FUNCTION_BLOCK Manual
VAR_INPUT
END_VAR

VAR_OUTPUT
END_VAR

VAR
	motorSelect: Multiplexer;
	EdgeDetectionRedButton: EdgeDetection;
	TIMER: TIMER;
	
	CountDown: CTUD;
	EdgeDetectionCD: BOOL;
	dropTimer: TON;
	rotateTimer: TON;
	stretchTimer: TON;
	clawTimer: TON;
	CounterDol: CTUD;
	visina: WORD;
	CounterCCW: CTUD;
	rotacija: WORD;
	CounterRazteg: CTUD;
	dolzina: WORD;
	CounterKlesce: CTUD;
	prijem: WORD;
	CounterVisina: CTUD;
END_VAR

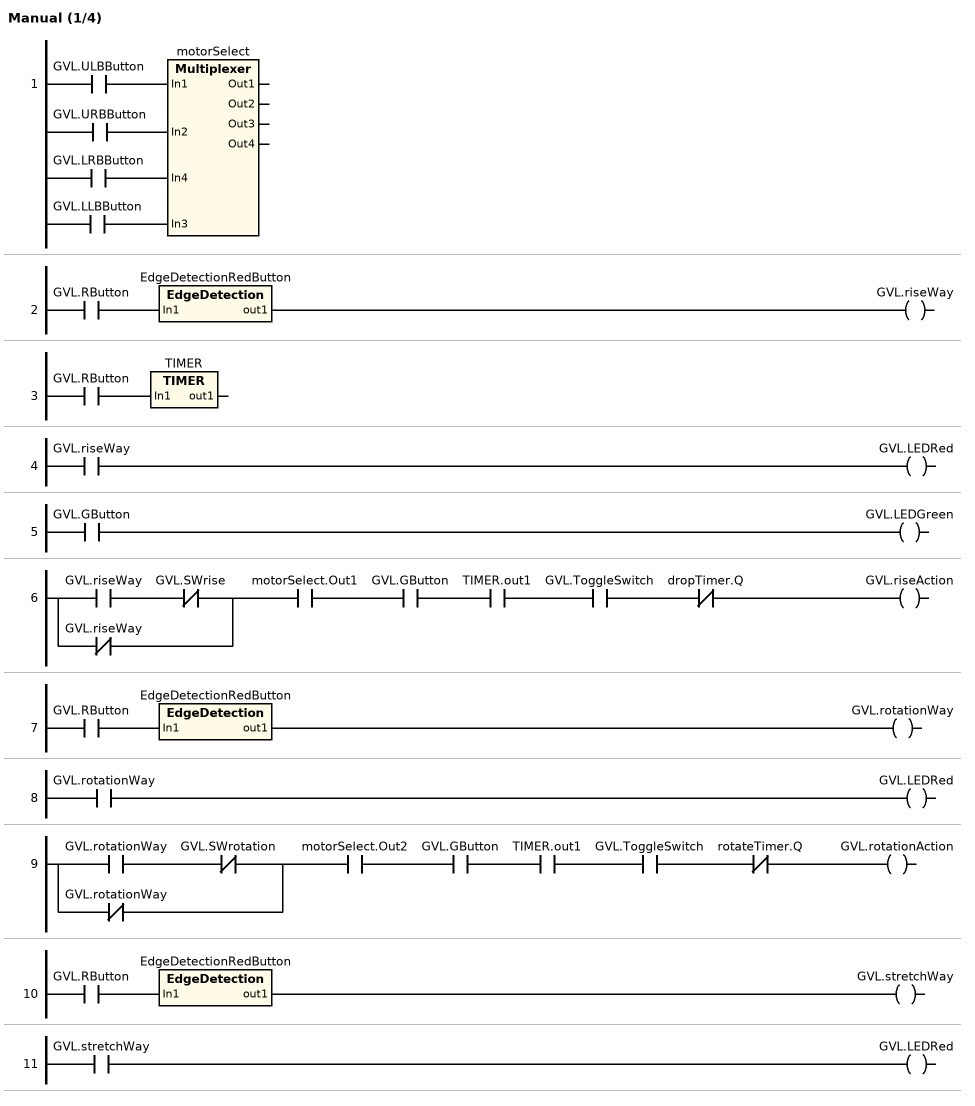
// NETWORK 1
motorSelect(In1 := GVL.ULBButton, In2 := GVL.URBButton, In4 := GVL.LRBButton, In3 := GVL.LLBButton); // Multiplexer

// NETWORK 2
EdgeDetectionRedButton(In1 := GVL.RButton); // EdgeDetection
GVL.riseWay := EdgeDetectionRedButton.out1;

// NETWORK 3
TIMER(In1 := GVL.RButton);

// NETWORK 4
GVL.LEDRed := GVL.riseWay;

// NETWORK 5
GVL.LEDGreen := GVL.GButton;

// NETWORK 6
GVL.riseAction := (GVL.riseWay AND NOT GVL.SWrise OR NOT GVL.riseWay) AND motorSelect.Out1 AND GVL.GButton AND TIMER.out1 AND GVL.ToggleSwitch AND NOT dropTimer.Q;

// NETWORK 7
EdgeDetectionRedButton(In1 := GVL.RButton); // EdgeDetection
GVL.rotationWay := EdgeDetectionRedButton.out1;

// NETWORK 8
GVL.LEDRed := GVL.rotationWay;

// NETWORK 9
GVL.rotationAction := (GVL.rotationWay AND NOT GVL.SWrotation OR NOT GVL.rotationWay) AND motorSelect.Out2 AND GVL.GButton AND TIMER.out1 AND GVL.ToggleSwitch AND NOT rotateTimer.Q;

// NETWORK 10
EdgeDetectionRedButton(In1 := GVL.RButton); // EdgeDetection
GVL.stretchWay := EdgeDetectionRedButton.out1;

// NETWORK 11
GVL.LEDRed := GVL.stretchWay;

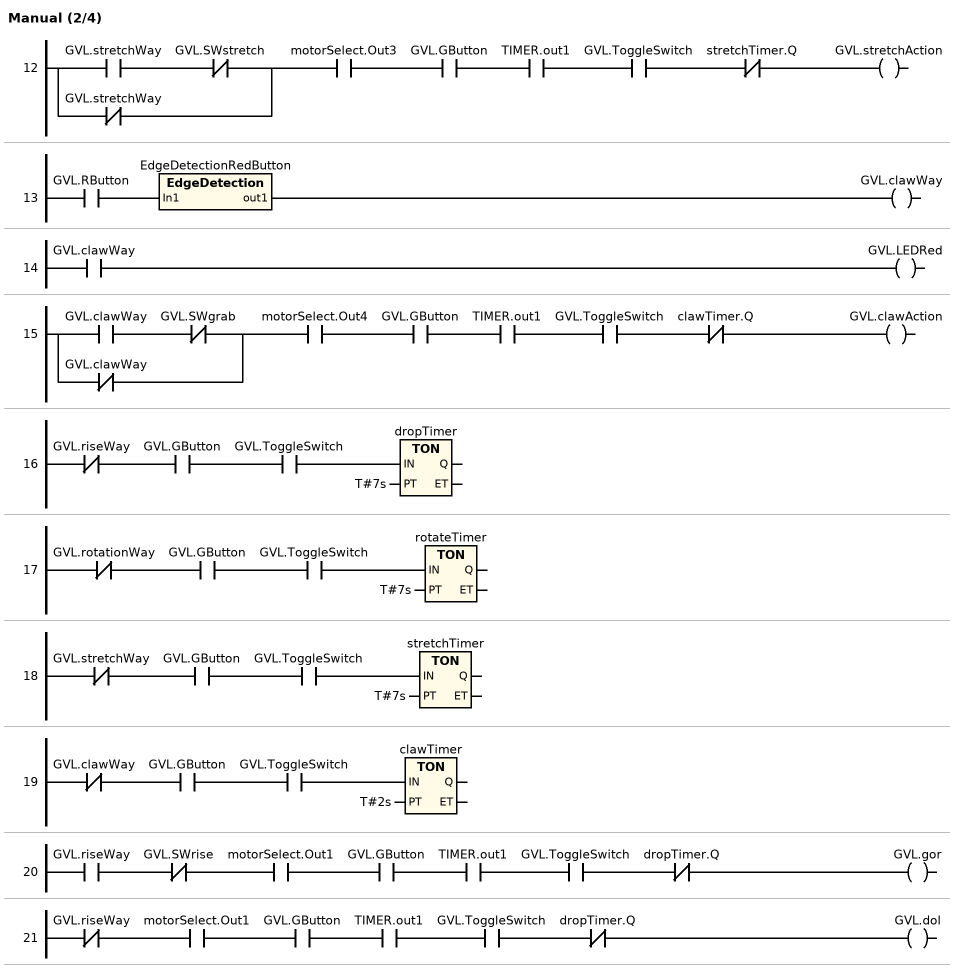
// NETWORK 12
GVL.stretchAction := (GVL.stretchWay AND NOT GVL.SWstretch OR NOT GVL.stretchWay) AND motorSelect.Out3 AND GVL.GButton AND TIMER.out1 AND GVL.ToggleSwitch AND NOT stretchTimer.Q;

// NETWORK 13
EdgeDetectionRedButton(In1 := GVL.RButton); // EdgeDetection
GVL.clawWay := EdgeDetectionRedButton.out1;

// NETWORK 14
GVL.LEDRed := GVL.clawWay;

// NETWORK 15
GVL.clawAction := (GVL.clawWay AND NOT GVL.SWgrab OR NOT GVL.clawWay) AND motorSelect.Out4 AND GVL.GButton AND TIMER.out1 AND GVL.ToggleSwitch AND NOT clawTimer.Q;

// NETWORK 16
dropTimer(IN := NOT GVL.riseWay AND GVL.GButton AND GVL.ToggleSwitch, PT := T#7s); // TON

// NETWORK 17
rotateTimer(IN := NOT GVL.rotationWay AND GVL.GButton AND GVL.ToggleSwitch, PT := T#7s); // TON

// NETWORK 18
stretchTimer(IN := NOT GVL.stretchWay AND GVL.GButton AND GVL.ToggleSwitch, PT := T#7s); // TON

// NETWORK 19
clawTimer(IN := NOT GVL.clawWay AND GVL.GButton AND GVL.ToggleSwitch, PT := T#2s); // TON

// NETWORK 20
GVL.gor := GVL.riseWay AND NOT GVL.SWrise AND motorSelect.Out1 AND GVL.GButton AND TIMER.out1 AND GVL.ToggleSwitch AND NOT dropTimer.Q;

// NETWORK 21
GVL.dol := NOT GVL.riseWay AND motorSelect.Out1 AND GVL.GButton AND TIMER.out1 AND GVL.ToggleSwitch AND NOT dropTimer.Q;

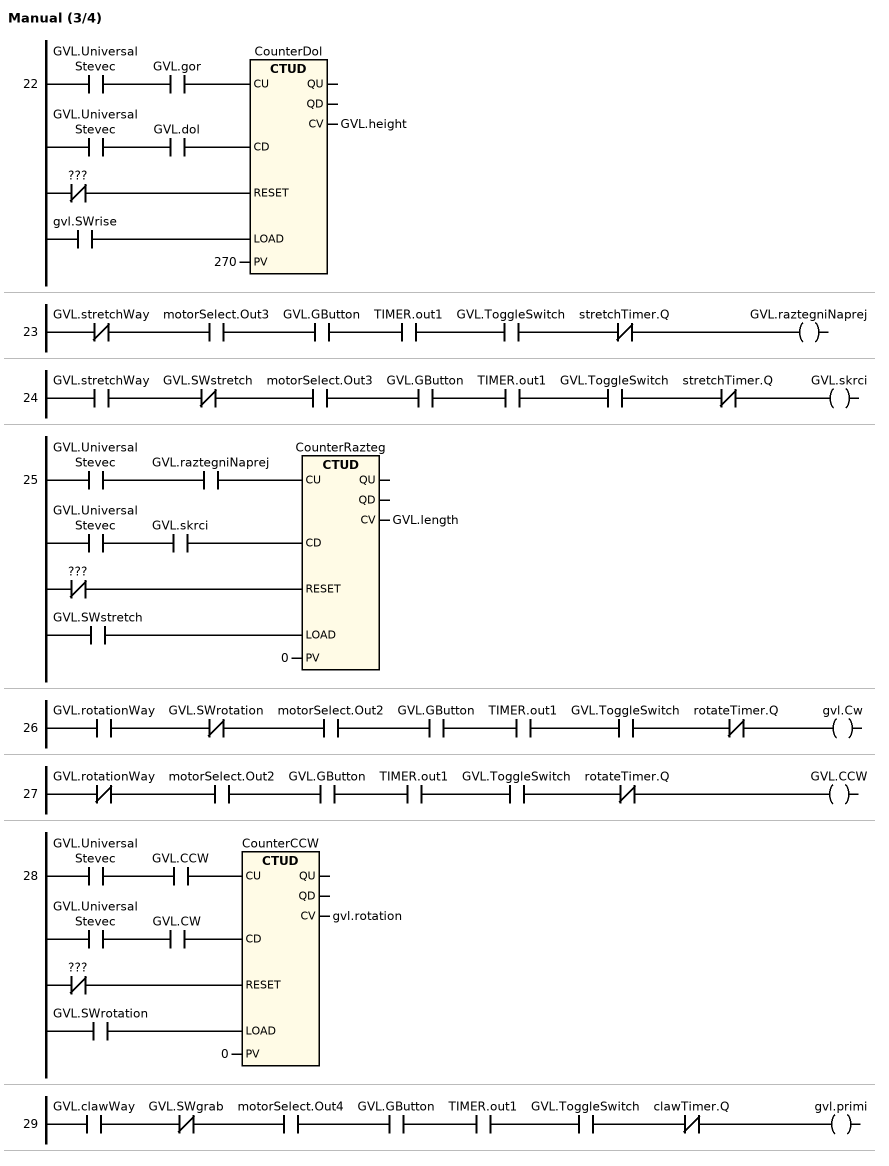
// NETWORK 22
CounterDol(
    CU := GVL.UniversalStevec AND GVL.gor,
    CD := GVL.UniversalStevec AND GVL.dol,
    LOAD := gvl.SWrise,
    PV := 270,
    CV => GVL.height); // CTUD

// NETWORK 23
GVL.raztegniNaprej := NOT GVL.stretchWay AND motorSelect.Out3 AND GVL.GButton AND TIMER.out1 AND GVL.ToggleSwitch AND NOT stretchTimer.Q;

// NETWORK 24
GVL.skrci := GVL.stretchWay AND NOT GVL.SWstretch AND motorSelect.Out3 AND GVL.GButton AND TIMER.out1 AND GVL.ToggleSwitch AND NOT stretchTimer.Q;

// NETWORK 25
CounterRazteg(
    CU := GVL.UniversalStevec AND GVL.raztegniNaprej,
    CD := GVL.UniversalStevec AND GVL.skrci,
    LOAD := GVL.SWstretch,
    PV := 0,
    CV => GVL.length); // CTUD

// NETWORK 26
gvl.Cw := GVL.rotationWay AND NOT GVL.SWrotation AND motorSelect.Out2 AND GVL.GButton AND TIMER.out1 AND GVL.ToggleSwitch AND NOT rotateTimer.Q;

// NETWORK 27
GVL.CCW := NOT GVL.rotationWay AND motorSelect.Out2 AND GVL.GButton AND TIMER.out1 AND GVL.ToggleSwitch AND NOT rotateTimer.Q;

// NETWORK 28
CounterCCW(
    CU := GVL.UniversalStevec AND GVL.CCW,
    CD := GVL.UniversalStevec AND GVL.CW,
    LOAD := GVL.SWrotation,
    PV := 0,
    CV => gvl.rotation); // CTUD

// NETWORK 29
gvl.primi := GVL.clawWay AND NOT GVL.SWgrab AND motorSelect.Out4 AND GVL.GButton AND TIMER.out1 AND GVL.ToggleSwitch AND NOT clawTimer.Q;

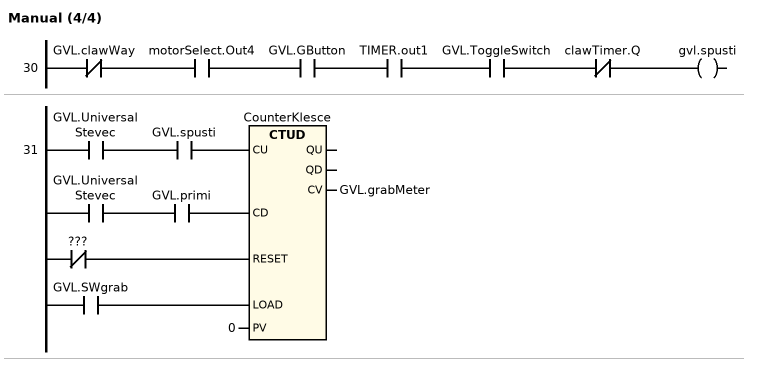
// NETWORK 30
gvl.spusti := NOT GVL.clawWay AND motorSelect.Out4 AND GVL.GButton AND TIMER.out1 AND GVL.ToggleSwitch AND NOT clawTimer.Q;

// NETWORK 31
CounterKlesce(
    CU := GVL.UniversalStevec AND GVL.spusti,
    CD := GVL.UniversalStevec AND GVL.primi,
    LOAD := GVL.SWgrab,
    PV := 0,
    CV => GVL.grabMeter); // CTUD

END_FUNCTION_BLOCK

(* stored: Version 1.1.0.1, ProductVersion 3.1.4024.15
   POU Manual: Id {8c93fc62-9243-4b19-bc29-a778beba09ad}, SpecialFunc None *)
